# EPICS autosave request: iocBoot/iocStdTest/auto_settings.req
file scalerSoftCtrl_settings.req P=xxx:,Q=scaler1:
